SUBAPPLICATION Uebung_022 (* Spiegelabfolge (2) *)
  (* Standard: 61499-2; Description: Copyright (c) 2023 Meisterschulen am Ostbahnhof This program and the accompanying materials are made available under the terms of the Eclipse Public License 2.0 which is available at https://www.eclipse.org/legal/epl-2.0/ SPDX-License-Identifier: EPL-2.0 *)
  (* Version 1.0, 2023-10-23, Franz Höpfinger, Meisterschulen am Ostbahnhof *)
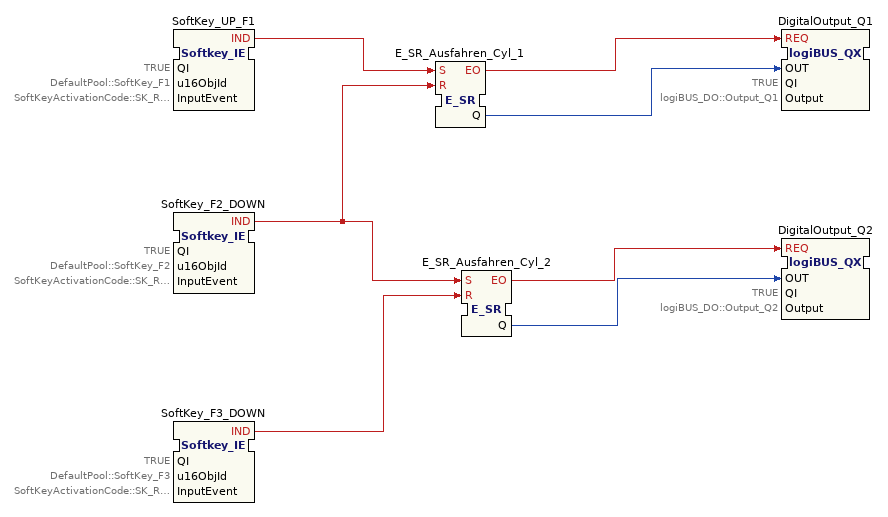
  (* START-Knopf *)
  (* Endlage Ausfahren_Cyl_1 *)
  (* Endlage Ausfahren_Cyl_2 *)
  (* Ausfahren_Cyl_1 *)
  (* Ausfahren_Cyl_2 *)
  FBS
    DigitalOutput_Q1 : logiBUS_QX(QI := TRUE, Output := logiBUS_DO::Output_Q1);
    SoftKey_UP_F1 : Softkey_IE(QI := TRUE, u16ObjId := DefaultPool::SoftKey_F1, InputEvent := SoftKeyActivationCode::SK_RELEASED);
    E_SR_Ausfahren_Cyl_1 : E_SR;
    SoftKey_F2_DOWN : Softkey_IE(QI := TRUE, u16ObjId := DefaultPool::SoftKey_F2, InputEvent := SoftKeyActivationCode::SK_RELEASED);
    DigitalOutput_Q2 : logiBUS_QX(QI := TRUE, Output := logiBUS_DO::Output_Q2);
    E_SR_Ausfahren_Cyl_2 : E_SR;
    SoftKey_F3_DOWN : Softkey_IE(QI := TRUE, u16ObjId := DefaultPool::SoftKey_F3, InputEvent := SoftKeyActivationCode::SK_RELEASED);
  END_FBS
  EVENT_CONNECTIONS
    SoftKey_UP_F1.IND TO E_SR_Ausfahren_Cyl_1.S;
    SoftKey_F2_DOWN.IND TO E_SR_Ausfahren_Cyl_1.R;
    E_SR_Ausfahren_Cyl_1.EO TO DigitalOutput_Q1.REQ;
    E_SR_Ausfahren_Cyl_2.EO TO DigitalOutput_Q2.REQ;
    SoftKey_F2_DOWN.IND TO E_SR_Ausfahren_Cyl_2.S;
    SoftKey_F3_DOWN.IND TO E_SR_Ausfahren_Cyl_2.R;
  END_CONNECTIONS
  DATA_CONNECTIONS
    E_SR_Ausfahren_Cyl_1.Q TO DigitalOutput_Q1.OUT;
    E_SR_Ausfahren_Cyl_2.Q TO DigitalOutput_Q2.OUT;
  END_CONNECTIONS
END_SUBAPPLICATION
